{attribute 'GeneratedUsingTerminal: EK1122-0000-0018'}
{attribute addProperty BoxType "EK1122-0000-0018"}
{attribute addProperty Id "Beckhoff_EJ1xxxsub_EK1100EK1100_1FC0878B2A_0001_EJ1100_0000_0018EJ1100_1FC0878B2A_0002_EJ1101_0022_0016EJ1101_7DD28DC43"}
{attribute addProperty CRC "871414933"}
{attribute addProperty Size "7"}
TYPE Beckhoff_EJ1xxxEK1122_33F0BC95 EXTENDS EK1122_1FC0878B :
STRUCT
	{attribute addProperty Name "Beckhoff_EJ1xxxsub_EK1100"}
	{attribute addProperty PreviousPort "Beckhoff EJ1xxxEK1122 : D"}
	Beckhoff_EJ1xxxsub_EK1100 : EK1100_1FC0878B;
	{attribute addProperty Name "A_0001_EJ1100_0000_0018"}
	{attribute addProperty PreviousPort "Beckhoff EJ1xxxsub EK1100 : C"}
	A_0001_EJ1100_0000_0018 : EJ1100_1FC0878B;
	{attribute addProperty Name "A_0002_EJ1101_0022_0016"}
	{attribute addProperty PreviousPort "A_0001(EJ1100-0000-0018) : C"}
	A_0002_EJ1101_0022_0016 : EJ1101_7DD28DC4;
END_STRUCT
END_TYPE

(* stored: Version 1.2.0.0, ProductVersion 3.1.4024.9
   DUT Beckhoff_EJ1xxxEK1122_33F0BC95: Id {64da6181-85cc-4a20-8a4a-538d301a4ecf} *)
